            TEST nBuffernummer
                CASE 1:
                    !
                    Incr nAantal_Balk1_In;
                      IF nAantal_Balk1_In = 8 THEN
                        Incr nAantal_Laag1_In;
                      ENDIF
                    Buffer_1_In;
                CASE 2:
                    !
                    Incr nAantal_Balk2_In;
                      IF nAantal_Balk2_In = 8 THEN
                        Incr nAantal_Laag2_In;
                      ENDIF
                    Buffer_2_In;
                CASE 3:
                    !
                    Incr nAantal_Balk3_In;
                      IF nAantal_Balk3_In = 8 THEN
                        Incr nAantal_Laag3_In;
                      ENDIF
                    Buffer_3_In;
                CASE 4:
                    !
                    Incr nAantal_Balk4_In;
                      IF nAantal_Balk4_In = 8 THEN
                        Incr nAantal_Laag4_In;
                      ENDIF
                    Buffer_4_In;
                CASE 5:
                    !
                    Incr nAantal_Balk5_In;
                      IF nAantal_Balk5_In = 8 THEN
                        Incr nAantal_Laag5_In;
                      ENDIF
                    Buffer_5_In;
                CASE 6:
                    !
                    Incr nAantal_Balk6_In;
                      IF nAantal_Balk6_In = 8 THEN
                        Incr nAantal_Laag6_In;
                      ENDIF
                    Buffer_6_In;
            ENDTEST
        ELSE
           RETURN;
        ENDIF

    ENDPROC

ENDMODULE
